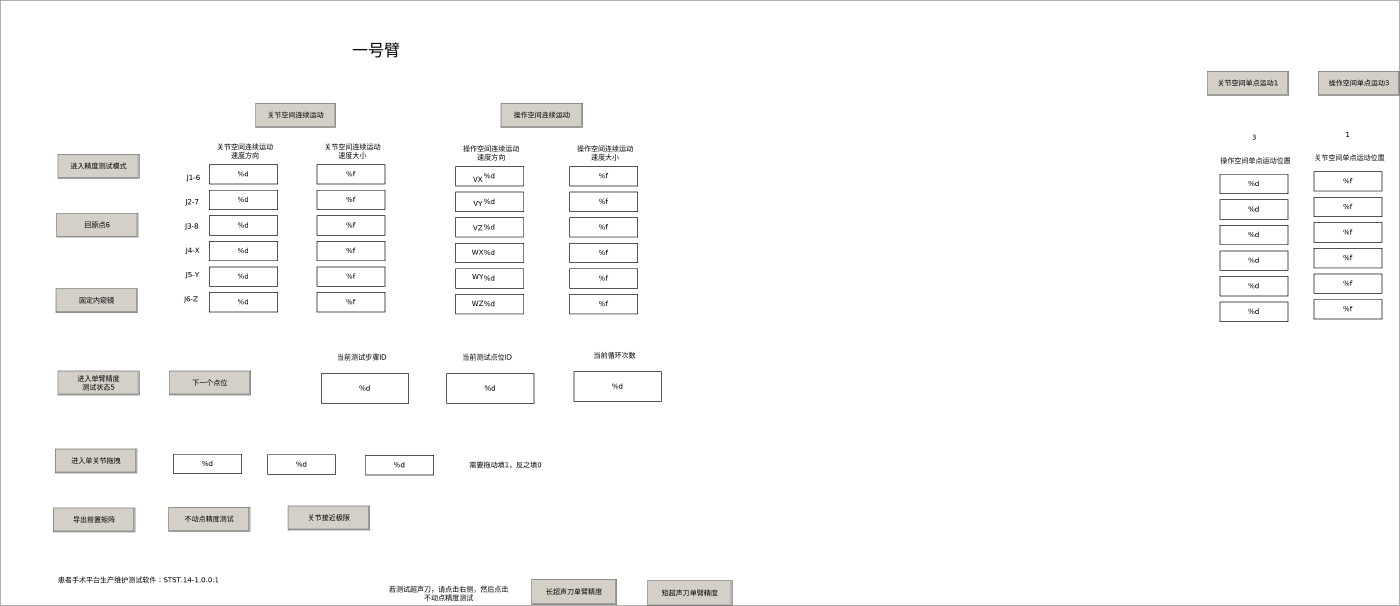
VISUALIZATION precision_a1  // 2189x948
    Label (513,57 150x43), "一号臂"
    Rectangle (327,257 107x31), "%d", text variable: g_motionTest.m_jntMotionDir[1][1]
        OnMouseClick: write the text variable via Default, min -1, max 1
    Label (308,222 150x29), "关节空间连续运动 速度方向"
    Rectangle (327,297 107x31), "%d", text variable: g_motionTest.m_jntMotionDir[1][2]
        OnMouseClick: write the text variable via Default, min -1, max 1
    Rectangle (327,337 107x31), "%d", text variable: g_motionTest.m_jntMotionDir[1][3]
        OnMouseClick: write the text variable via Default, min -1, max 1
    Rectangle (327,377 107x31), "%d", text variable: g_motionTest.m_jntMotionDir[1][4]
        OnMouseClick: write the text variable via Default, min -1, max 1
    Rectangle (327,417 107x31), "%d", text variable: g_motionTest.m_jntMotionDir[1][5]
        OnMouseClick: write the text variable via Default, min -1, max 1
    Rectangle (327,457 107x31), "%d", text variable: g_motionTest.m_jntMotionDir[1][6]
        OnMouseClick: write the text variable via Default, min -1, max 1
    Rectangle (2054,268 107x31), "%f", text variable: g_motionTest.m_targetJntPos[1][1]
        OnMouseClick: write the text variable via Default
    Label (2035,232 150x30), "关节空间单点运动位置"
    Rectangle (2054,308 107x31), "%f", text variable: g_motionTest.m_targetJntPos[1][2]
        OnMouseClick: write the text variable via Default
    Rectangle (2054,348 107x31), "%f", text variable: g_motionTest.m_targetJntPos[1][3]
        OnMouseClick: write the text variable via Default
    Rectangle (2054,388 107x31), "%f", text variable: g_motionTest.m_targetJntPos[1][4]
        OnMouseClick: write the text variable via Default
    Rectangle (2054,428 107x31), "%f", text variable: g_motionTest.m_targetJntPos[1][5]
        OnMouseClick: write the text variable via Default
    Rectangle (2054,468 107x31), "%f", text variable: g_motionTest.m_targetJntPos[1][6]
        OnMouseClick: write the text variable via Default
    Label (2032,196 150x30), "1"
    Rectangle (495,257 107x31), "%f", text variable: g_motionTest.m_jntVel[1][1]
        OnMouseClick: write the text variable via Default
    Label (476,222 150x29), "关节空间连续运动 速度大小"
    Rectangle (495,297 107x31), "%f", text variable: g_motionTest.m_jntVel[1][2]
        OnMouseClick: write the text variable via Default
    Rectangle (495,337 107x31), "%f", text variable: g_motionTest.m_jntVel[1][3]
        OnMouseClick: write the text variable via Default
    Rectangle (495,377 107x31), "%f", text variable: g_motionTest.m_jntVel[1][4]
        OnMouseClick: write the text variable via Default
    Rectangle (495,417 107x31), "%f", text variable: g_motionTest.m_jntVel[1][5]
        OnMouseClick: write the text variable via Default
    Rectangle (495,457 107x31), "%f", text variable: g_motionTest.m_jntVel[1][6]
        OnMouseClick: write the text variable via Default
    Rectangle (1907,272 107x31), "%d"
    Label (1888,237 150x29), "操作空间单点运动位置"
    Rectangle (1907,312 107x31), "%d"
    Rectangle (1907,352 107x31), "%d"
    Rectangle (1907,392 107x31), "%d"
    Rectangle (1907,432 107x31), "%d"
    Rectangle (1907,472 107x31), "%d"
    Label (1886,200 150x30), "3"
    Rectangle (712,260 107x31), "%d", text variable: g_motionTest.m_spatialMotionDir[1][1]
        OnMouseClick: write the text variable via Default, min -1, max 1
    Label (693,225 150x29), "操作空间连续运动 速度方向"
    Rectangle (712,300 107x31), "%d", text variable: g_motionTest.m_spatialMotionDir[1][2]
        OnMouseClick: write the text variable via Default, min -1, max 1
    Rectangle (712,340 107x31), "%d", text variable: g_motionTest.m_spatialMotionDir[1][3]
        OnMouseClick: write the text variable via Default, min -1, max 1
    Rectangle (712,380 107x31), "%d", text variable: g_motionTest.m_spatialMotionDir[1][4]
        OnMouseClick: write the text variable via Default, min -1, max 1
    Rectangle (712,420 107x31), "%d", text variable: g_motionTest.m_spatialMotionDir[1][5]
        OnMouseClick: write the text variable via Default, min -1, max 1
    Rectangle (712,460 107x31), "%d", text variable: g_motionTest.m_spatialMotionDir[1][6]
        OnMouseClick: write the text variable via Default, min -1, max 1
    Rectangle (890,260 107x31), "%f", text variable: g_motionTest.m_spatialVel[1][1]
        OnMouseClick: write the text variable via Default
    Label (871,225 150x29), "操作空间连续运动 速度大小"
    Rectangle (890,300 107x31), "%f", text variable: g_motionTest.m_spatialVel[1][2]
        OnMouseClick: write the text variable via Default
    Rectangle (890,340 107x31), "%f", text variable: g_motionTest.m_spatialVel[1][3]
        OnMouseClick: write the text variable via Default
    Rectangle (890,380 107x31), "%f", text variable: g_motionTest.m_spatialVel[1][4]
        OnMouseClick: write the text variable via Default
    Rectangle (890,420 107x31), "%f", text variable: g_motionTest.m_spatialVel[1][5]
        OnMouseClick: write the text variable via Default
    Rectangle (890,460 107x31), "%f", text variable: g_motionTest.m_spatialVel[1][6]
        OnMouseClick: write the text variable via Default
    Button (90,241 128x38), "进入精度测试模式", colour toggle: g_motionTest.m_enterPrecisionTestMode[1]
        toggle g_motionTest.m_enterPrecisionTestMode[1]
    Group (1887,111 302x38), invisible if: TRUE
        Button (0,0 128x38), "关节空间单点运动1", colour toggle: g_motionTest.m_uiArmModeL[1,1]
            tap g_motionTest.m_uiArmMode[1,1]
        Button (174,0 128x38), "操作空间单点运动3", colour toggle: g_motionTest.m_uiArmModeL[1,3]
            tap g_motionTest.m_uiArmMode[1,3]
    Button (399,161 126x38), "关节空间连续运动", colour toggle: g_motionTest.m_uiArmModeL[1,2]
        tap g_motionTest.m_uiArmMode[1,2]
    Button (783,161 128x38), "操作空间连续运动", colour toggle: g_motionTest.m_uiArmModeL[1,4]
        tap g_motionTest.m_uiArmMode[1,4]
    Button (88,333 128x38), "回原点6", colour toggle: g_motionTest.m_uiArmModeL[1,6]
        tap g_motionTest.m_uiArmMode[1,6]
    Button (90,580 128x38), "进入单臂精度 测试状态5", colour toggle: g_motionTest.m_uiArmMode[1,5]
        toggle g_motionTest.m_uiArmMode[1,5]
    Button (264,580 128x38), "下一个点位", colour toggle: g_motionTest.m_nextStep[1]
        tap g_motionTest.m_nextStep[1]
    Rectangle (502,584 137x47), "%d", text variable: g_motionTest.m_curStep[1]
    Label (491,544 150x30), "当前测试步骤ID"
    Rectangle (698,584 137x47), "%d", text variable: g_motionTest.m_testPointId[1]
    Label (687,544 150x30), "当前测试点位ID"
    Rectangle (897,581 137x47), "%d", text variable: g_motionTest.m_testCycleId[1]
    Label (886,541 150x30), "当前循环次数"
    Label (287,263 31x30), "J1-6"
    Label (277,301 47x30), "J2-7"
    Label (282,339 36x30), "J3-8"
    Label (281,377 41x30), "J4-X"
    Label (281,415 40x30), "J5-Y"
    Label (281,453 36x30), "J6-Z"
    Group (672,266 26x224)
        Label (0,0 150x30), "VX"
        Label (0,38 150x30), "VY"
        Label (0,76 150x30), "VZ"
        Label (0,114 150x30), "WX"
        Label (0,152 150x30), "WY"
        Label (0,194 150x30), "WZ"
    Rectangle (271,710 107x31), "%d", text variable: g_motionTest.m_dragJntFlag[1][1]
        OnMouseClick: write the text variable via Default, min -1, max 1
    Button (86,702 128x38), "进入单关节拖拽", colour toggle: g_motionTest.m_uiArmMode[1,7]
        toggle g_motionTest.m_uiArmMode[1,7]
    Rectangle (418,711 107x31), "%d", text variable: g_motionTest.m_dragJntFlag[1][2]
        OnMouseClick: write the text variable via Default, min -1, max 1
    Rectangle (571,712 107x31), "%d", text variable: g_motionTest.m_dragJntFlag[1][3]
        OnMouseClick: write the text variable via Default, min -1, max 1
    Label (707,713 167x29), "需要拖动填1，反之填0"
    Button (83,794 128x38), "导出前置矩阵"
        tap g_motionTest.m_writeData[1]
    Button (263,793 128x38), "不动点精度测试", colour toggle: g_motionTest.m_uiArmMode[1,8]
        toggle g_motionTest.m_uiArmMode[1,8]
    Button (450,791 128x38), "关节接近极限", colour toggle: g_motionTest.m_jntOutFlag[1]
    Button (831,906 133x40), "长超声刀单臂精度", colour toggle: g_motionTest.m_UltrasoundKnife_Long[1]
        toggle g_motionTest.m_UltrasoundKnife_Long[1]
    Button (1012,908 133x40), "短超声刀单臂精度", colour toggle: g_motionTest.m_UltrasoundKnife_Short[1]
        toggle g_motionTest.m_UltrasoundKnife_Short[1]
    Label (602,914 199x29), "若测试超声刀，请点击右侧，然后点击不动点精度测试"
    Label (79,891 275x33), "患者手术平台生产维护测试软件：STST.14-1.0.0.1"
    Button (87,451 128x38), "固定内窥镜", colour toggle: g_motionTest.m_uiFixedEndoFlag
        toggle g_motionTest.m_uiFixedEndoFlag
END_VISUALIZATION

(* stored: Version 1.1.0.1, ProductVersion 3.1.4024.11
   Visu precision_a1: Id {c275d056-9c8b-436c-b15b-86e3d9a625b0} *)
